FUNCTION_BLOCK FB_Transor
VAR_INPUT
  
END_VAR
VAR_OUTPUT
END_VAR
VAR_IN_OUT
	IOdwCtrl : DWORD;
END_VAR
VAR
  iChan : SINT; // Kanalnummer im IOdwState
  
	// %I / %Q ********************
	QbTransor       AT %Q* : BOOL;

END_VAR



QbTransor := GETBIT32(IOdwCtrl, iChan);

// end of functionblock

PROPERTY PUBLIC PiChannel : SINT
SET

IF (PiChannel >= 0) AND (PiChannel <= 31) THEN
  iChan := PiChannel;
ELSE
  iChan := 0;
END_IF
END_SET
END_PROPERTY

END_FUNCTION_BLOCK

(* stored: Version 1.1.0.1, ProductVersion 3.1.4018.10
   POU FB_Transor: Id {88a34746-49b1-4be7-affd-e82147f46edf}, SpecialFunc None
   Property PiChannel: Id {312a05a4-0fef-4dc4-9242-a3bf1e37eddf}
   Set Set: Id {82cb4133-60df-4239-9a37-03479ce73626} *)
